FUNCTION_BLOCK FB_ElmoGDCBellCoE
VAR_IN_OUT
	stCoE	:	ST_ElmoGDCBellCoEParams;
END_VAR
VAR_INPUT
END_VAR
VAR_OUTPUT
END_VAR
VAR
	fbCoERead	:	FB_CoERead_ByDriveRef;
	// To make up for not having a .bDone output
	ftCoeReadBusy: F_TRIG;
	CaseVar: INT := 1;
	udiIP	:	UDINT;
	uiChecksum	:	UDINT;

	pTempPointer : POINTER TO REAL;
	fTempFloat : REAL;
END_VAR
VAR CONSTANT
	c5VSupply : ST_CoEIndSub := (nIndex:=16#2206, nSubIndex:=0);
	cDriveTemp : ST_CoEIndSub := (nIndex:=16#22A3, nSubIndex:=1);
	cIP : ST_CoEIndSub := (nIndex:=16#1111, nSubIndex:=1);
	cParamChksm	:	ST_CoEIndSub := (nIndex:=16#2060, nSubIndex:=0);
END_VAR

(* A. Wallace 17-3-22
ElmoMC Gold DC Bell CoE Read


This FB cyclically reads CoE Parameters from the ElmoMC drives.
*)

CASE CaseVar OF
	
1:
//Drive temperature
fbCoERead.nIndex := cDriveTemp.nIndex;
fbCoERead.nSubIndex := cDriveTemp.nSubIndex;
fbCoERead.pDstBuf := ADR(stCoE.uiDriveTemp);
fbCoERead.cbBufLen := SIZEOF(stCoE.uiDriveTemp);
pTempPointer := fbCoERead.pDstBuf;
fTempFloat := pTempPointer^;
2:
//5v supply
fbCoERead.nIndex := c5vSupply.nIndex;
fbCoERead.nSubIndex := c5vSupply.nSubIndex;
fbCoERead.pDstBuf := ADR(stCoE.ui5VSupply);
fbCoERead.cbBufLen := SIZEOF(stCoE.ui5VSupply);
3:
//Parameter checksum
fbCoERead.nIndex := cParamChksm.nIndex;
fbCoERead.nSubIndex := cParamChksm.nSubIndex;
fbCoERead.pDstBuf := ADR(uiChecksum);
fbCoERead.cbBufLen := SIZEOF(uiChecksum);
stCoE.testChecksum := UDINT_TO_DINT(uiChecksum);
4:
//IP
fbCoERead.nIndex := cIP.nIndex;
fbCoERead.nSubIndex := cIP.nSubIndex;
fbCoERead.pDstBuf := ADR(udiIP);
fbCoERead.cbBufLen := SIZEOF(udiIP);
END_CASE


fbCoERead.bExecute := TRUE;
ftCoeReadBusy(CLK:=fbCoERead.bBusy);
IF ftCoeReadBusy.Q THEN
	fbCoERead.bExecute := FALSE;
	//<TODO> check for errors
	IF NOT fbCoERead.bError THEN
		//Switch to the other case
		CaseVar := CaseVar + 1;
		IF CaseVar > 3 THEN CaseVar := 1; END_IF
	ELSE
		;
	END_IF
END_IF

ACT_CoEReadFB();

ACTION ACT_CoEReadFB:
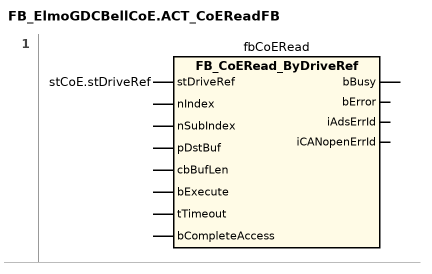
// NETWORK 1
fbCoERead(stDriveRef := stCoE.stDriveRef); // FB_CoERead_ByDriveRef
END_ACTION

END_FUNCTION_BLOCK

(* stored: Version 1.1.0.1, ProductVersion 3.1.4022.18
   POU FB_ElmoGDCBellCoE: Id {91acbbac-f6fe-4d79-9df9-4139d2e826f8}, SpecialFunc None
   Action ACT_CoEReadFB: Id {854d3f04-b0de-4b54-adaa-712dc279dab2} *)
